(* PLC project Generated.project, CODESYS CODESYS V3.5 SP19 Patch 1 *)
(* stored: creationDateTime 2026-09-06T13:00:42.534858, modificationDateTime 2026-09-06T13:00:42.534858 *)

(* ═══════════════════════════════════════════════════════════════ 🕹️ ST_AcquisitionJoystickQualified — Données joystick qualifiées ─────────────────────────────────────────────────────────────── 🎯 Rôle : Encapsuler les commandes d'axes, statut homme-mort et diagnostics produits par FB_Joystick dans PRG_02_Acquisition. 📤 Producteur unique : PRG_02_Acquisition (Data.Joystick). 📄 Doc : DOC/AF/AF_Partie-06_Acquisition_Qualification_IO_v2.4.md ═══════════════════════════════════════════════════════════════ *)
TYPE ST_AcquisitionJoystickQualified : STRUCT
  AxisX : ST_fbJoystick_AxisCmd;  (* 📊 Commande et direction qualifiée axe X *)
  AxisY : ST_fbJoystick_AxisCmd;  (* 📊 Commande et direction qualifiée axe Y *)
  DeadmanArmed : BOOL;  (* 🔒 Homme-mort armé et valide *)
  AtNeutralXY : BOOL;  (* 🟢 Les deux axes X et Y sont au neutre *)
  ArmingPermitDenied : BOOL;  (* ⚠️ Tentative d'armement sans permission *)
  Ready : BOOL;  (* 🟢 Façade joystick prête et opérationnelle *)
  Fault : ST_Fault;  (* ❌ Diagnostic défaut joystick *)
  NeutralXAct : INT;  (* 📍 Valeur ADC neutre calibré X *)
  NeutralYAct : INT;  (* 📍 Valeur ADC neutre calibré Y *)
END_STRUCT;
END_TYPE

(* ======================================================================= 🧩 ST_Fault — Brique socle défaut (2 vues : live + latchée) ─────────────────────────────────────────────────────────────── 🎯 Rôle : porter l'état défaut d'un composant, applicable dans TOUS les cas (acquittable ou non), sans brique warning séparée. • Vue LIVE (Error / ErrorId) : suit la cause, retombe seule à 0. • Vue LATCHÉE (Latched / LatchedId): mémorisée au défaut, reste jusqu'au front Reset. Le choix acquittable / non-acquittable se fait PAR CAUSE (ST_FaultCause.Latching), jamais par bloc. 🔒 Sécurité : interlock TOUJOURS sur la cause brute (Error / ErrorId), jamais sur l'acquittement. Reset TOUJOURS effectif, jamais conditionné (std §9). 🧬 Composition : brique de base réutilisable — sortie de FB, struct métier, GVL. Texte IHM NON stocké ici : dérivé côté IHM depuis LatchedId / ErrorId. 📄 Doc : DOC/STDS/CODE_QUALITY_STANDARDS.md §2quinquies / §9 ======================================================================= *)
TYPE ST_Fault : STRUCT
  Error : BOOL;  (* <-- [DIAG] vue LIVE : au moins une cause présente maintenant *)
  ErrorId : WORD;  (* <-- [DIAG] bitfield des causes présentes maintenant (0 si aucune) *)
  Latched : BOOL;  (* <-- [DIAG] vue LATCHÉE : défaut non acquitté, reste jusqu'au front Reset *)
  LatchedId : WORD;  (* <-- [DIAG] ErrorId figé à l'apparition du défaut, effacé au Reset *)
END_STRUCT;
END_TYPE

(* ======================================================================= 🕹️ ST_fbJoystick_AxisCmd — Consigne d'axe normalisée (sortie FB_Joystick) ─────────────────────────────────────────────────────────────── 🎯 Rôle : Structure de consigne d'axe produite par FB_Joystick. 📤 Champs : Enable, StartStop, SpeedTgt (%) + StepTgt (palier 1..5) + direction en bits (DirectionPositive/Negative, AtNeutral). SpeedTgt reste pour l'IHM, StepTgt pour la logique. 📄 Doc métier : DOC/AF/AF_Partie-08_Fonction_Joystick_v2.5.md ======================================================================= *)
TYPE ST_fbJoystick_AxisCmd : STRUCT
  Enable : BOOL;  (* === CONSIGNES DE PILOTAGE AXE === --> [CMD] Autorisation globale pipeline (FALSE=neutralisation, sorties coupees) *)
  StartStop : BOOL;  (* --> [CMD] Validation de mouvement (TRUE=acceleration, FALSE=deceleration/arret) *)
  SpeedTgt : REAL;  (* --> [CMD] Vitesse cible non signee (0...100 %, signe/sens donné par Direction) - IHM *)
  StepTgt : INT;  (* --> [CMD] Palier de vitesse (1..5, 0=arret) - logique/limitations (derive de SpeedTgt) *)
  DirectionNegative : BOOL;  (* --> [CMD] Direction joystick ou intension de gestuelle *)
  DirectionPositive : BOOL;  (* --> [CMD] Direction joystick ou intension de gestuelle *)
  AtNeutral : BOOL;  (* --> [CMD] TRUE si axes en zone morte (position centrale) *)
  Direction : INT;  (* === MONITORING IHM (derive des bits ci-dessus, jamais lu en interlock) === <-- [STAT] Sens -1=Rev / 0=Neutre / +1=Fwd (anim IHM fleche ; lu aussi logique treuils PRG_04) *)
  Deflection : INT;  (* <-- [STAT] Deflexion signee -100..+100 % (anim IHM jauge/barre) *)
END_STRUCT;
END_TYPE
